(* IEC 61131-3 sources: Mirroring_Webvisu/graph/visu/Processing, 11 files *)

(* ---- GVL_Data.GVL ---- *)
{attribute 'qualified_only'}
VAR_GLOBAL
    rVisuTemperature : REAL;
    dtVisuTimestamp : DT;
    sVisuTimestampString : STRING(255); // String version for easier binding if needed
END_VAR

(* ---- DirCreate.st ---- *)
FUNCTION DirCreate : BOOL
VAR_INPUT
    sDirectoryPath : STRING(255);   // Full path of directory to create
END_VAR
VAR
    result : RTS_IEC_RESULT;        // Result code
END_VAR

// Create the directory
result := SysDirCreate(
    szDir := sDirectoryPath,
    pResult := ADR(result)
);

// Return TRUE if directory was created successfully
IF result = 0 THEN  // ERR_OK
    DirCreate := TRUE;
ELSE
    DirCreate := FALSE;
END_IF

(* ---- FileCopy.st ---- *)
FUNCTION FileCopy : BOOL
VAR_INPUT
    sSourceFile : STRING(255);      // Full path to source file
    sDestDirectory : STRING(255);   // Destination directory path
    sDestFileName : STRING(255);    // Destination file name
END_VAR
VAR
    sDestPath : STRING(255);        // Complete destination path
    result : RTS_IEC_RESULT;        // Result code
END_VAR

// Build complete destination path
sDestPath := CONCAT(sDestDirectory, '\');
sDestPath := CONCAT(sDestPath, sDestFileName);

// Copy the file
result := SysFileCopy(
    szFileDest := sDestPath,
    szFileSource := sSourceFile,
    pResult := ADR(result)
);

// Return TRUE if copy was successful
IF result = 0 THEN  // ERR_OK
    FileCopy := TRUE;
ELSE
    FileCopy := FALSE;
END_IF

(* ---- FileExist.st ---- *)
FUNCTION FileExist : BOOL
VAR_INPUT
    sFilePath : STRING(255);    // Full path to the file to check
END_VAR
VAR
    hFile : RTS_IEC_HANDLE;     // File handle
    result : RTS_IEC_RESULT;    // Result code
END_VAR
VAR CONSTANT
    INVALID_HANDLE : RTS_IEC_HANDLE := 16#FFFFFFFF;
END_VAR

// Try to open the file in read mode
hFile := SysFileOpen(
    szFile := sFilePath,
    am := ACCESS_MODE.AM_READ,
    pResult := ADR(result)
);

// Check if file was opened successfully
IF hFile <> INVALID_HANDLE THEN
    // File exists, close it
    SysFileClose(hFile := hFile);
    FileExist := TRUE;
ELSE
    // File does not exist or cannot be opened
    FileExist := FALSE;
END_IF

(* ---- FB_DirectoryReader.st ---- *)
FUNCTION_BLOCK FB_DirectoryReader
VAR_INPUT
    xExecute : BOOL;                    // Rising edge triggers directory read
    sDirectoryPath : STRING(255);       // Path to directory to read
END_VAR

VAR_OUTPUT
    xDone : BOOL;                       // TRUE when reading is complete
    xBusy : BOOL;                       // TRUE while reading is in progress
    xError : BOOL;                      // TRUE if an error occurred
    eErrorID : RTS_IEC_RESULT;         // Error code if xError is TRUE
    udiFileCount : UDINT;              // Number of files found
    aFileList : ARRAY[0..99] OF STRING(255);  // List of file names found
END_VAR

VAR
    // Internal state machine
    eState : (IDLE, OPEN_DIR, READ_ENTRIES, CLOSE_DIR, DONE, ERROR);
    xExecuteOld : BOOL;

    // SysDir function blocks and variables
    hDir : RTS_IEC_HANDLE;             // Directory handle
    sDirEntry : STRING(255);           // Current directory entry name
    dirInfo : DirInfo;                 // Directory information structure
    result : RTS_IEC_RESULT;           // Result code

    // Internal index
    udiIndex : UDINT;                  // Current index in file list
END_VAR

VAR CONSTANT
    INVALID_HANDLE : RTS_IEC_HANDLE := 16#FFFFFFFF;
END_VAR

// Implementation
// Detect rising edge on xExecute
IF xExecute AND NOT xExecuteOld THEN
    eState := OPEN_DIR;
    xDone := FALSE;
    xBusy := TRUE;
    xError := FALSE;
    eErrorID := 0;
    udiFileCount := 0;
    udiIndex := 0;
END_IF
xExecuteOld := xExecute;

CASE eState OF
    IDLE:
        xBusy := FALSE;
        xDone := FALSE;

    OPEN_DIR:
        // Open the directory
        hDir := SysDirOpen(
            szDir := sDirectoryPath,
            szDirEntry := sDirEntry,
            diMaxDirEntry := SIZEOF(sDirEntry),
            pDirInfo := ADR(dirInfo),
            pResult := ADR(result)
        );

        IF hDir <> INVALID_HANDLE THEN
            // Directory opened successfully
            eState := READ_ENTRIES;
        ELSE
            // Failed to open directory
            xError := TRUE;
            eErrorID := result;
            eState := ERROR;
        END_IF

    READ_ENTRIES:
        // Read next directory entry
        result := SysDirRead(
            hDir := hDir,
            szDirEntry := sDirEntry,
            diMaxDirEntry := SIZEOF(sDirEntry),
            pDirInfo := ADR(dirInfo)
        );

        IF result = 0 THEN  // ERR_OK
            // Successfully read an entry
            // Check if it's a file (not a directory)
            IF dirInfo.diDirectory = 0 THEN  // Not a directory
                // Store file name in array if space available
                IF udiIndex < 100 THEN
                    aFileList[udiIndex] := sDirEntry;
                    udiIndex := udiIndex + 1;
                    udiFileCount := udiFileCount + 1;
                END_IF
            END_IF
            // Continue reading next entry

        ELSIF result = 16#00000002 THEN  // ERR_END_OF_DIR
            // Reached end of directory
            eState := CLOSE_DIR;

        ELSE
            // Error reading directory
            xError := TRUE;
            eErrorID := result;
            eState := CLOSE_DIR;  // Still try to close the directory
        END_IF

    CLOSE_DIR:
        // Close the directory handle
        result := SysDirClose(hDir := hDir);

        IF xError THEN
            eState := ERROR;
        ELSE
            eState := DONE;
        END_IF

    DONE:
        xBusy := FALSE;
        xDone := TRUE;
        eState := IDLE;

    ERROR:
        xBusy := FALSE;
        xDone := TRUE;
        eState := IDLE;
END_CASE

(* ---- MemAggregation.st ---- *)
TYPE E_TimeSpan :
(
    LAST_15M := 0,
    LAST_30M,
    LAST_1H,
    LAST_6H,
    LAST_12H,
    LAST_24H,
    LAST_48H
);
END_TYPE

TYPE E_AggType :
(
    AGG_AVERAGE := 0,
    AGG_MEDIAN
);
END_TYPE

FUNCTION_BLOCK FB_MemAggregation
VAR_INPUT
    xExecute : BOOL; // Cycle pulse (e.g. 1s)
    rInput : REAL;
    eTimeSpan : E_TimeSpan := E_TimeSpan.LAST_15M;
    eAggType : E_AggType := E_AggType.AGG_AVERAGE;
    xReset : BOOL;
END_VAR
VAR_OUTPUT
    rResult : REAL;
    xReady : BOOL; // Buffer is sufficiently filled
    udiCurrentCount : UDINT;
END_VAR
VAR
    // Ring Buffer (Max size for 1h/1s or 48h/1min = 3600 + overhead)
    // 48h * 60m = 2880 pts. 1h * 3600s = 3600 pts. Max is 3600.
    aRingBuffer : ARRAY[0..3599] OF REAL;
    udiHead : UDINT := 0; // Write Index
    udiCount : UDINT := 0; // Current items in buffer

    // Minute Downsampling Buffer
    aMinuteBuffer : ARRAY[0..59] OF REAL;
    udiMinIndex : UDINT := 0;

    // Configuration
    udiTargetSize : UDINT;
    xDownsample : BOOL; // TRUE if we aggregate 1s -> 1min

    // Internal
    xInitialized : BOOL;
    rSum : REAL;
    i : UDINT;
    j : UDINT;
    rTemp : REAL;
    aSortBuffer : ARRAY[0..3599] OF REAL; // For median sorting
    udiSortCount : UDINT;
END_VAR

// Reset Logic
IF xReset THEN
    udiHead := 0;
    udiCount := 0;
    udiMinIndex := 0;
    rResult := 0;
    xReady := FALSE;
    xInitialized := FALSE;
END_IF

// Configuration Setup (Run once or on change)
IF NOT xInitialized THEN
    CASE eTimeSpan OF
		E_TimeSpan.LAST_15M: udiTargetSize := 900;  xDownsample := FALSE; // 1s
		E_TimeSpan.LAST_30M: udiTargetSize := 1800; xDownsample := FALSE; // 1s
		E_TimeSpan.LAST_1H:  udiTargetSize := 3600; xDownsample := FALSE; // 1s
		E_TimeSpan.LAST_6H:  udiTargetSize := 360;  xDownsample := TRUE;  // 1min (360pts)
		E_TimeSpan.LAST_12H: udiTargetSize := 720;  xDownsample := TRUE;  // 1min (720pts)
		E_TimeSpan.LAST_24H: udiTargetSize := 1440; xDownsample := TRUE;  // 1min (1440pts)
		E_TimeSpan.LAST_48H: udiTargetSize := 2880; xDownsample := TRUE;  // 1min (2880pts)
    ELSE
        udiTargetSize := 900; xDownsample := FALSE;
    END_CASE
    xInitialized := TRUE;
END_IF

// Input Processing (On Execute Rising/High?)
// Assuming xExecute is a pulse every second.
IF xExecute THEN

    IF xDownsample THEN
        // Collect into minute buffer
        IF udiMinIndex < 60 THEN
            aMinuteBuffer[udiMinIndex] := rInput;
            udiMinIndex := udiMinIndex + 1;
        END_IF

        // If minute full, calculate avg and push to Ring
        IF udiMinIndex >= 60 THEN
            rSum := 0;
            FOR i := 0 TO 59 DO
                rSum := rSum + aMinuteBuffer[i];
            END_FOR

            rTemp := rSum / 60.0;

            // PUSH to Ring
            aRingBuffer[udiHead] := rTemp;
            udiHead := udiHead + 1;
            IF udiHead >= udiTargetSize THEN
                udiHead := 0;
            END_IF
            IF udiCount < udiTargetSize THEN
                udiCount := udiCount + 1;
            END_IF

            // Reset Minute Buffer
            udiMinIndex := 0;
        END_IF
    ELSE
        // Direct Push (1s resolution)
        aRingBuffer[udiHead] := rInput;
        udiHead := udiHead + 1;
        IF udiHead >= udiTargetSize THEN
            udiHead := 0;
        END_IF
        IF udiCount < udiTargetSize THEN
            udiCount := udiCount + 1;
        END_IF
    END_IF

    // Calculate Final Result (Aggregated over Ring Buffer)
    // NOTE: For performance, Average could be optimized 'Rolling'.
    // Here we recalculate full buffer for simplicity/robustness.

    IF udiCount > 0 THEN
        IF eAggType = E_AggType.AGG_AVERAGE THEN
            // Calculate Average
            rSum := 0;
            FOR i := 0 TO udiCount - 1 DO
                rSum := rSum + aRingBuffer[i];
            END_FOR
            rResult := rSum / UDINT_TO_REAL(udiCount);

        ELSIF eAggType = E_AggType.AGG_MEDIAN THEN
            // Calculate Median (Expensive: Sort required)
            // Copy to sort buffer
            // SysMemCpy(ADR(aSortBuffer), ADR(aRingBuffer), ...);
            // Manual copy to be safe
            FOR i := 0 TO udiCount - 1 DO
                aSortBuffer[i] := aRingBuffer[i];
            END_FOR

            // Bubble Sort (Simple, but O(N^2). 3600^2 is huge.
            // Should be used carefully. Maybe optimized sort or standard lib sort?)
            // Keeping it simple for prototype. Warning: Cycle time!
            // Optimization: If performance is issue, use 'Running Median' approx or partial sort.

            udiSortCount := udiCount;
            FOR i := 0 TO udiSortCount - 2 DO
                FOR j := 0 TO udiSortCount - i - 2 DO
                    IF aSortBuffer[j] > aSortBuffer[j+1] THEN
                         rTemp := aSortBuffer[j];
                         aSortBuffer[j] := aSortBuffer[j+1];
                         aSortBuffer[j+1] := rTemp;
                    END_IF
                END_FOR
            END_FOR

            // Pick middle
            IF (udiSortCount MOD 2) <> 0 THEN
                // Odd: Middle element
                rResult := aSortBuffer[udiSortCount / 2];
            ELSE
                // Even: Avg of two middle
                rResult := (aSortBuffer[udiSortCount / 2] + aSortBuffer[(udiSortCount / 2) - 1]) / 2.0;
            END_IF
        END_IF
    ELSE
        rResult := 0;
    END_IF

    xReady := (udiCount >= udiTargetSize);
    udiCurrentCount := udiCount;

END_IF

// --------------------------------------------------------------------------
// Helper Method: PUSH to Ring Buffer
// We can't use 'METHOD' in simple ST file export unless structured correctly.
// We'll use inline code or internal Action if available.
// For ST file compatibility, I will just inline the logic above or call it via Action?
// No, standard ST expects FUNCTION_BLOCK to contain everything in body or methods.
// I used MEM_PUSH call above - I need to implement it or inline it.
// I will convert "MEM_PUSH(val)" to inline logic above.
// --------------------------------------------------------------------------

(* ---- ReadCSV.st ---- *)
FUNCTION_BLOCK FB_ReadCSV
VAR_INPUT
    xExecute : BOOL;
    sFileName : STRING(255);
END_VAR
VAR_OUTPUT
    xDone : BOOL;
    xBusy : BOOL;
    xError : BOOL;
    dwErrorID : RTS_IEC_RESULT;
    aFileLines : ARRAY[0..99] OF STRING(255);
    udiLineCount : UDINT;
END_VAR
VAR
    iState : INT := 0;
    xExecuteOld : BOOL;
    hFile : RTS_IEC_HANDLE := RTS_INVALID_HANDLE;
    sBaseDir : STRING(255) := '/home/codesys/';
    sFullPath : STRING(255);

    // Reading buffers
    byReadChar : BYTE;
    sCurrentLine : STRING(255);
    ulBytesRead : UDINT;
    iLineIndex : INT;

    // Helpers
    pDest : POINTER TO BYTE;
    byNull : BYTE := 0;
END_VAR
VAR CONSTANT
    RTS_INVALID_HANDLE : RTS_IEC_HANDLE := 16#FFFFFFFF;
END_VAR

// Edge detection
IF xExecute AND NOT xExecuteOld THEN
    xDone := FALSE;
    xBusy := TRUE;
    xError := FALSE;
    dwErrorID := 0;
    udiLineCount := 0;
    iState := 10;

    // Clear previous results
    FOR iLineIndex := 0 TO 99 DO
        aFileLines[iLineIndex] := '';
    END_FOR
END_IF
xExecuteOld := xExecute;

// State machine
CASE iState OF
    10: // Open File
        // Construct full path
        sFullPath := CONCAT(sBaseDir, sFileName);

        // Open in Read mode
        hFile := SysFileOpen(szFile := sFullPath, am := ACCESS_MODE.AM_READ, pResult := ADR(dwErrorID));

        IF hFile <> RTS_INVALID_HANDLE THEN
            iState := 20;
            sCurrentLine := '';
            udiLineCount := 0;
        ELSE
            xError := TRUE;
            xBusy := FALSE;
            iState := 0;
        END_IF

    20: // Read Loop
        // Read 1 byte
        ulBytesRead := SysFileRead(
            hFile := hFile,
            pbyBuffer := ADR(byReadChar),
            ulSize := 1,
            pResult := ADR(dwErrorID)
        );

        IF ulBytesRead = 0 THEN
            // EOF reached
            // Save last line if not empty
            IF LEN(sCurrentLine) > 0 AND udiLineCount < 100 THEN
                aFileLines[udiLineCount] := sCurrentLine;
                udiLineCount := udiLineCount + 1;
            END_IF
            iState := 30; // Close file

        ELSE
            // Process character
            IF byReadChar = 16#0A THEN // LF (Line Feed)
                // End of line found
                // Note: CR (16#0D) might be present at end of string, we can trim it or just leave it depending on usage.

                // Remove CR if previous char was CR (simple check: if last char of sCurrentLine is $R)
                // Actually easier: just ignore CR when building string, OR handle LF as terminator.

                IF udiLineCount < 100 THEN
                    aFileLines[udiLineCount] := sCurrentLine;
                    udiLineCount := udiLineCount + 1;
                END_IF
                sCurrentLine := ''; // Reset buffer

            ELSIF byReadChar = 16#0D THEN // CR (Carriage Return)
                // Ignore CR, wait for LF
                ;
            ELSE
                // Append character
                // Safety check for max length
                IF LEN(sCurrentLine) < 255 THEN
                    // Calculate append position
                    pDest := ADR(sCurrentLine) + LEN(sCurrentLine);

                    // Copy character
                    SysMemCpy(
                        pDest := pDest,
                        pSrc := ADR(byReadChar),
                        udiCount := 1
                    );

                    // Null terminate next byte
                    SysMemCpy(
                        pDest := pDest + 1,
                        pSrc := ADR(byNull),
                        udiCount := 1
                    );
                END_IF
            END_IF
        END_IF

    30: // Close File
        SysFileClose(hFile := hFile);
        hFile := RTS_INVALID_HANDLE;

        IF NOT xError THEN
            xDone := TRUE;
        END_IF
        xBusy := FALSE;
        iState := 0;

END_CASE

(* ---- WriteCSV.st ---- *)
FUNCTION_BLOCK FB_WriteCSV
VAR_INPUT
    xExecute : BOOL;
    sFileName : STRING(255);
    sHeader : STRING(255);
    sDataLine : STRING(255);
    tWriteInterval : TIME := T#60S; // Default 60s interval
    xAddNewline : BOOL := TRUE;
END_VAR
VAR_OUTPUT
    xDone : BOOL;
    xBusy : BOOL;
    xError : BOOL;
    dwErrorID : RTS_IEC_RESULT;
END_VAR
VAR
    xExecuteOld : BOOL;
    hFile : RTS_IEC_HANDLE := RTS_INVALID_HANDLE;
    sBaseDir : STRING(255) := '/home/codesys/';
    sFullPath : STRING(255);
    sWriteBuffer : STRING(255);
    ulBytesWritten : UDINT;
    xFileExisted : BOOL;

    // Buffer Variables
    aBuffer : ARRAY[0..199] OF STRING(255);
    udiBufferCount : UDINT := 0;
    fbFlushTimer : TON;
    i : UDINT; // Loop counter
END_VAR
VAR CONSTANT
    RTS_INVALID_HANDLE : RTS_IEC_HANDLE := 16#FFFFFFFF;
    MAX_BUFFER_SIZE : UDINT := 200;
END_VAR

// 1. Handle Input (Buffering)
IF xExecute AND NOT xExecuteOld THEN
    xBusy := TRUE;
    xDone := FALSE;
    xError := FALSE;

    IF udiBufferCount < MAX_BUFFER_SIZE THEN
        aBuffer[udiBufferCount] := sDataLine;
        udiBufferCount := udiBufferCount + 1;
    ELSE
        // Buffer Overflow - Optional: Trigger immediate flush or Error?
        // We will trigger immediate flush below.
        ;
    END_IF
END_IF
xExecuteOld := xExecute;

// 2. Timer Logic
// Timer runs if there is data in buffer
fbFlushTimer(IN := udiBufferCount > 0, PT := tWriteInterval);

// 3. Flush Condition
IF (fbFlushTimer.Q OR udiBufferCount >= MAX_BUFFER_SIZE) AND udiBufferCount > 0 THEN
    // Perform Synchronous Flush

    // A. Create Directory (Once check)
    // We could do this only once, but safety first.
    SysDirCreate(szDir := sBaseDir);

    // B. Open File
    sFullPath := CONCAT(sBaseDir, sFileName);

    xFileExisted := FileExist(sFilePath := sFullPath);

    IF xFileExisted THEN
         hFile := SysFileOpen(szFile := sFullPath, am := ACCESS_MODE.AM_APPEND, pResult := ADR(dwErrorID));
    ELSE
         hFile := SysFileOpen(szFile := sFullPath, am := ACCESS_MODE.AM_WRITE, pResult := ADR(dwErrorID));
    END_IF

    IF hFile <> RTS_INVALID_HANDLE THEN

        // C. Write Header (If new)
        IF NOT xFileExisted AND LEN(sHeader) > 0 THEN
            sWriteBuffer := sHeader;
            IF xAddNewline THEN
                sWriteBuffer := CONCAT(sWriteBuffer, '$R$N');
            END_IF
            SysFileWrite(hFile := hFile, pbyBuffer := ADR(sWriteBuffer), ulSize := LEN(sWriteBuffer), pResult := ADR(dwErrorID));
        END_IF

        // D. Write Buffer Data
        FOR i := 0 TO udiBufferCount - 1 DO
            sWriteBuffer := aBuffer[i];
            IF xAddNewline THEN
                sWriteBuffer := CONCAT(sWriteBuffer, '$R$N');
            END_IF

            SysFileWrite(hFile := hFile, pbyBuffer := ADR(sWriteBuffer), ulSize := LEN(sWriteBuffer), pResult := ADR(dwErrorID));

            // Check error? If error, maybe stop?
            // For now continue and flag error at end.
            IF dwErrorID <> 0 THEN
                xError := TRUE;
            END_IF
        END_FOR

        // E. Close File
        SysFileClose(hFile := hFile);
        hFile := RTS_INVALID_HANDLE;

        // F. Reset Buffer
        IF NOT xError THEN
            udiBufferCount := 0;
            xDone := TRUE;
        END_IF
    ELSE
        xError := TRUE;
    END_IF

    xBusy := FALSE; // Pulse Busy off after flush? Or keep Busy while buffering?
    // Usually Busy=True means "Processing". Buffering is "Processing".
    // Let's reset Busy only after flush or if buffer is empty.
    // If we just buffered, we are technically "Waiting".
    // Let's pulse xDone when Flush is complete.
END_IF

// Reset Done trigger (optional, usually valid for one cycle)
// If we want xDone to stay TRUE until next Execute?
// Standard FB: xDone valid when Job Completed.
// Here "Job" is "Append to Buffer" OR "Flush"?
// Let's say xDone is TRUE when Buffer Added? Or when Flushed?
// "Support bulk writing... single process".
// User likely checks log to see if "written".
// With buffering, "Written" effectively means "Buffered".
// So let's set xDone := TRUE immediately after buffering,
// AND maybe a separate output xFlushed?
// Or stick to simple logic: xDone implies "Handled".
// I will keep xDone = TRUE after Flush.
// Note: If I don't set xDone after Buffering, the user might hang waiting for it.
// CHANGE: Set xDone := TRUE after Buffering successfully.
// The Flush is an internal maintenance task.
// If Flush fails, xError becomes TRUE.

IF xExecute AND NOT xError THEN
   xDone := TRUE; // Data accepted into buffer
   xBusy := FALSE;
END_IF

(* ---- Example_MemAggregation.st ---- *)
PROGRAM Example_MemAggregation
VAR
    fbAgg : FB_MemAggregation;
    rSensorVal : REAL := 20.0;
    rAggResult : REAL;

    // Test Signal Generation
    fbTimer : TON := (PT := T#1S); // 1s trigger
    xTrigger : BOOL;

    // Configuration
    eSetSpan : E_TimeSpan := E_TimeSpan.LAST_15M;
    eSetAgg : E_AggType := E_AggType.AGG_AVERAGE;
END_VAR

// 1s Update Loop (Simulates cyclic task)
fbTimer(IN := NOT fbTimer.Q);
IF fbTimer.Q THEN
    xTrigger := TRUE;

    // Simulate Noise/Change
    rSensorVal := rSensorVal + 0.1;
    IF rSensorVal > 30.0 THEN rSensorVal := 20.0; END_IF
ELSE
    xTrigger := FALSE;
END_IF

// Call Aggregation
fbAgg(
    xExecute := xTrigger,
    rInput := rSensorVal,
    eTimeSpan := eSetSpan,
    eAggType := eSetAgg,
    xReset := FALSE
);

// Read Result
rAggResult := fbAgg.rResult;

// Note: rResult updates every time xExecute triggers (every 1s).
// For 15M, it updates immediately.
// For 6H (1min resolution), it updates the Ring Buffer only once per minute,
// so rResult might stay stable until next minute update?
// No, the logic calculates average of EXISTING buffer each cycle.
// So it stays stable until buffer changes.

(* ---- Example_ReadCSV.st ---- *)
PROGRAM Example_ReadCSV
VAR
    fbReadCSV : FB_ReadCSV;
    xTriggerRead : BOOL;
    aMyData : ARRAY[0..99] OF STRING(255);
    udiCount : UDINT;
END_VAR

// Call the Function Block
fbReadCSV(
    xExecute := xTriggerRead,
    sFileName := 'log.csv'
);

// Capture results when done
IF fbReadCSV.xDone THEN
    aMyData := fbReadCSV.aFileLines;
    udiCount := fbReadCSV.udiLineCount;
    xTriggerRead := FALSE;
END_IF

// Handle Error
IF fbReadCSV.xError THEN
    xTriggerRead := FALSE;
END_IF

(* ---- Example_WriteCSV.st ---- *)
PROGRAM Example_WriteCSV
VAR
    fbWriteCSV : FB_WriteCSV;
    xTriggerWrite : BOOL;

    // Aggregation Blocks
    fbAggHum : FB_MemAggregation;
    fbAggTemp : FB_MemAggregation;
    fbAggPress : FB_MemAggregation;

    // Data String
    sMyData : STRING(255);
    sCSVHeader : STRING(255) := 'Timestamp,Humidity_Avg,Temperature_Avg,Pressure_Avg';

    // Simulated Sensor Data
    rHumidity : REAL := 45.0;
    rTemperature : REAL := 22.5;
    rPressure : REAL := 1013.0;
    dtNow : DT := DT#2023-10-27-10:00:00;
    stLocal_TimeStamp : SysTime;

    // Timer for generating data (Fast: 100ms)
    fbDataTimer : TON := (PT := T#100MS);

    iCount : INT := 0;

	// time
	stLocal_TimeStamp : SysTime;

END_VAR

dtNow := TO_DT(stLocal_TimeStamp / TIME_TO_ULINT(TIME#1MS)); // DT#2018-6-6-10:24:54
// Trigger write every 100ms
fbDataTimer(IN := NOT fbDataTimer.Q);
IF fbDataTimer.Q THEN
    xTriggerWrite := TRUE;

    // Simulate changing data (Noise)
    rHumidity := rHumidity + 0.1;
    IF rHumidity > 60 THEN rHumidity := 45; END_IF

    rTemperature := rTemperature + 0.05;
    IF rTemperature > 30 THEN rTemperature := 20; END_IF

    rPressure := rPressure + 0.2;
    IF rPressure > 1020 THEN rPressure := 1000; END_IF

    // Update Aggregators (e.g. LAST_15M Average)
    fbAggHum(xExecute := TRUE, rInput := rHumidity, eTimeSpan := E_TimeSpan.LAST_15M, eAggType := E_AggType.AGG_AVERAGE);
    fbAggTemp(xExecute := TRUE, rInput := rTemperature, eTimeSpan := E_TimeSpan.LAST_15M, eAggType := E_AggType.AGG_AVERAGE);
    fbAggPress(xExecute := TRUE, rInput := rPressure, eTimeSpan := E_TimeSpan.LAST_15M, eAggType := E_AggType.AGG_AVERAGE);

    // Format Data using RAW Sensor Data
    sCSVHeader := 'Timestamp,Humidity,Temperature,Pressure';

    sMyData := DT_TO_STRING(dtNow);
    sMyData := CONCAT(sMyData, ',');
    sMyData := CONCAT(sMyData, REAL_TO_STRING(rHumidity));
    sMyData := CONCAT(sMyData, ',');
    sMyData := CONCAT(sMyData, REAL_TO_STRING(rTemperature));
    sMyData := CONCAT(sMyData, ',');
    sMyData := CONCAT(sMyData, REAL_TO_STRING(rPressure));

    // Update GVL for Visualization
    GVL_Data.rVisuTemperature := rTemperature;
    GVL_Data.dtVisuTimestamp := dtNow;
    GVL_Data.sVisuTimestampString := DT_TO_STRING(dtNow);

ELSE
    // Reset Execute pulse for Aggregators (if needed, but xExecute := TRUE above acts as pulse if in IF block?)
    // Actually standard FB usually needs FALSE then TRUE for edge?
    // FB_MemAggregation checks "IF xExecute THEN".
    // If we call it only inside IF fbDataTimer.Q, it is TRUE for that cycle.
    // But we MUST call FBs cyclically if they have internal state management that needs it?
    // FB_MemAggregation strictly acts "IF xExecute THEN". So calling it only on trigger is fine IF we don't need it to do anything else (like internal timers).
    // Our FB_MemAggregation doesn't have internal timers, just buffer logic.
    // So calling it inside the IF block is acceptable for this logic.
    ;
END_IF

// Call the CSV Writer
// Buffer data every time xTriggerWrite is True (every 100ms)
fbWriteCSV(
    xExecute := xTriggerWrite,
    sFileName := 'sensor_log.csv',
    sHeader := sCSVHeader,
    sDataLine := sMyData,
    tWriteInterval := T#60S,
    xAddNewline := TRUE
);

// Reset trigger immediately
IF xTriggerWrite THEN
    xTriggerWrite := FALSE;
END_IF
